(* PLC project v0.6.04_CycleSemiAuto.project, CODESYS CODESYS V3.5 SP19 Patch 1 *)
(* stored: creationDateTime 2026-08-01T01:07:33.347380, modificationDateTime 2026-08-01T01:07:33.347380 *)

TYPE ST_Winch_SymmetryData : STRUCT
  DeltaStartDelay_Ms, DeltaBrakeReleaseTime_Ms, DeltaBrakeApplyTime_Ms : UDINT;
  DeltaStopDistance_Mm, DeltaStopTime_Ms : UDINT;
  MaxSyncDeviation_M : REAL;
END_STRUCT;
END_TYPE
